Universal Robots PolyScope program: g01_apply.urp

Program g01_apply (installation=default directory=/programs createdIn=5.9.1.1031110 lastSavedIn=5.9.1.1031110 robotSerialNumber=20195501059)
Calibrated DH parameters: a=[0.000146, -0.418764, -0.053981, 0.000058, -0.000023, 0]; d=[0.162545, 37.319448, -206.067439, 168.881546, 0.09955, 0.099464]; alpha=[1.57004, -0.001979, 0.002304, 1.570607, -1.57066, 0]; deltaTheta=[0, -0.174616, -1.258233, 1.432844, -0.000001, 0]
Robot Program (runOnlyOnce=false)
  MoveL speed 250 mm/s, acceleration 1200 mm/s^2 (useActiveTCP=true) feature=Base
    Waypoint approach_bolt: TCP in base x=221.242 y=-344.604 z=215.619 mm, rx=-0.1092 ry=-2.9553 rz=-0.7196 rad; joints [102.684, -85.041, 99.258, -76.331, 271.455, -343.446] deg; TCP offset x=0 y=0 z=158 mm, rx=0 ry=0 rz=0 rad
    MoveDirectionNode (selectedDirection=ZPlus toolParams=0.02, 1.2) feature=Joint_6_name
      Until TOOL_CONTACT_DETECTION (allowActions=true retraction=0 decelerationAcceleration=3 decelerationAngularAcceleration=34.906585)
        Force Frame feature=Joint_6_name; selection=[0, 0, 1, 0, 0, 1]; wrench=[0, 0, 10, 0, 0, 1]; limitsForce=[0.15, 0.15, 0.01, 1.047198, 1.047198, 1.047198]; limitsMotion=[0.1, 0.1, 0.1, 0.349066, 0.349066, 0.349066]
          Wait Sleep waitTime=10
        URCap Gripper (Robotiq_Grippers, Robotiq Inc.) dataModel(position=59.29411764705882, force=100.0, speed=100.0, positionInDouble=59.29411764705882, forceInDouble=100.0, speedInDouble=100.0, slaveIds=[9], blocking=true)
        MoveDirectionNode (selectedDirection=ZMinus) feature=Joint_6_name
          Until DISTANCE (allowActions=false deceleration=3 distanceNodeType=STOP) Distance=0.05; motionParameters(blendRadius=0)
      Until DISTANCE (allowActions=true deceleration=3 distanceNodeType=STOP) Distance=0.025; motionParameters(blendRadius=0)
        Halt
